{attribute 'GeneratedUsingTerminal: EK1122-0000-0018'}
{attribute addProperty BoxType "EK1122-0000-0018"}
{attribute addProperty Id "Beckhoff_EL19xxsub_EK1100EK1100_1FC0878B2"}
{attribute addProperty CRC "719697273"}
{attribute addProperty Size "2"}
TYPE Beckhoff_EL19xxEK1122_2AE5B579 EXTENDS EK1122_1FC0878B :
STRUCT
	{attribute addProperty Name "Beckhoff_EL19xxsub_EK1100"}
	{attribute addProperty PreviousPort "Beckhoff EL19xxEK1122 : D"}
	Beckhoff_EL19xxsub_EK1100 : EK1100_1FC0878B;
END_STRUCT
END_TYPE

(* stored: Version 1.2.0.0, ProductVersion 3.1.4024.9
   DUT Beckhoff_EL19xxEK1122_2AE5B579: Id {71a2f72c-05f8-4955-9581-8652ec9947bc} *)
